FUNCTION shiftLeft : ARRAY[0..99] OF REAL
VAR_INPUT
	inputbuffer : ARRAY[0..99] OF REAL;
END_VAR
VAR
	tempIndex : UINT := 0;
	tempbuffer : ARRAY[0..99] OF REAL;
END_VAR

FOR tempIndex := 0 TO 98 DO
	tempbuffer[tempIndex] := inputbuffer[tempIndex+1];
END_FOR

shiftleft := tempbuffer;
RETURN;

END_FUNCTION

(* stored: Version 1.1.0.1, ProductVersion 3.1.4024.13
   POU shiftLeft: Id {4936dee2-6a18-416e-9168-89c328cbbc30}, SpecialFunc None *)
